// TIA Portal V17 export
// export: Created 2024-08-07T21:43:58.427102Z, ExportSetting WithDefaults, DisplayName Totally Integrated Automation Portal, DisplayVersion V17 Update 7, DisplayName TIA Portal Openness, DisplayVersion V17 Update 7, DisplayName TIA Portal Version Control Interface, DisplayVersion V17, DisplayName SINAMICS Startdrive Advanced, DisplayVersion V17 SP2, DisplayName SINAMICS Startdrive G110M, G120, G120C, G120D, G120P, G115D, DisplayVersion V17 SP2, DisplayName SINAMICS Startdrive G130, G150, S120, S150, SINAMICS MV, S210, DisplayVersion V17 SP2, DisplayName STEP 7 Professional, DisplayVersion V17 Update 7, DisplayName STEP 7 Safety, DisplayVersion V17 Update 6, DisplayName WinCC Advanced / Unified PC, DisplayVersion V17 Update 7
FUNCTION_BLOCK "READER_LOGIC"   // FB24, LAD
{ S7_Optimized_Access := 'TRUE' }
VERSION : 0.1
// stored: AutoNumber true, IsIECCheckEnabled false, IsRetainMemResEnabled false, MemoryReserve 100, SetENOAutomatically false, UDAEnableTagReadback false
   VAR_INPUT
      MODE : UInt;
      INIT_SCAN : Bool;
      SCAN_BUSY : Bool;
      SCAN_COMPLETE : Bool;
      STA_REC_1 : Bool;
      STA_REC : Bool;
      SCAN_OK1 : Bool;
      SCAN_OK2 : Bool;
      IJC_DISABLE : Bool;
      SCAN_LABEL : String;
      SCAN_POSITION : Int;
      SCAN_LEN : Int;
      READ_OF_SCAN : HW_SUBMODULE;
      NUM_OF_TUBE : Bool;
      RESET_SCANER : Bool;
   END_VAR
   VAR_OUTPUT
      REQUEST_SCAN : Bool;
      READ_STRG : String;
      SCAN_OK : Bool;
      MSG_STATUS_REQ : Bool;
      NFP_AUX : String;
      NFP_AUX2 : String;
      LECTURA_SCANER_ST : String;
      SCAN_CLEAR : Bool;
   END_VAR
   VAR
      RET_TRIG : IEC_TIMER;
   END_VAR
   VAR_TEMP
      ERROR_RECIBIDO_ESCANER : Int;
      RECIBIDO_SCANER : Array[0..254] of Char;
      RECIBIDO_SCANER_STRG : String;
      LECTURA_SCANER : String;
      done : Bool;
   END_VAR
   VAR_TEMP   // added for the SCL form of the ladder/FBD networks
      _w1 : Bool;
      _w2 : Bool;
      _w3 : Bool;
      _w4 : Bool;
      _w5 : Bool;
      _w6 : Bool;
   END_VAR
BEGIN

REGION Network 1
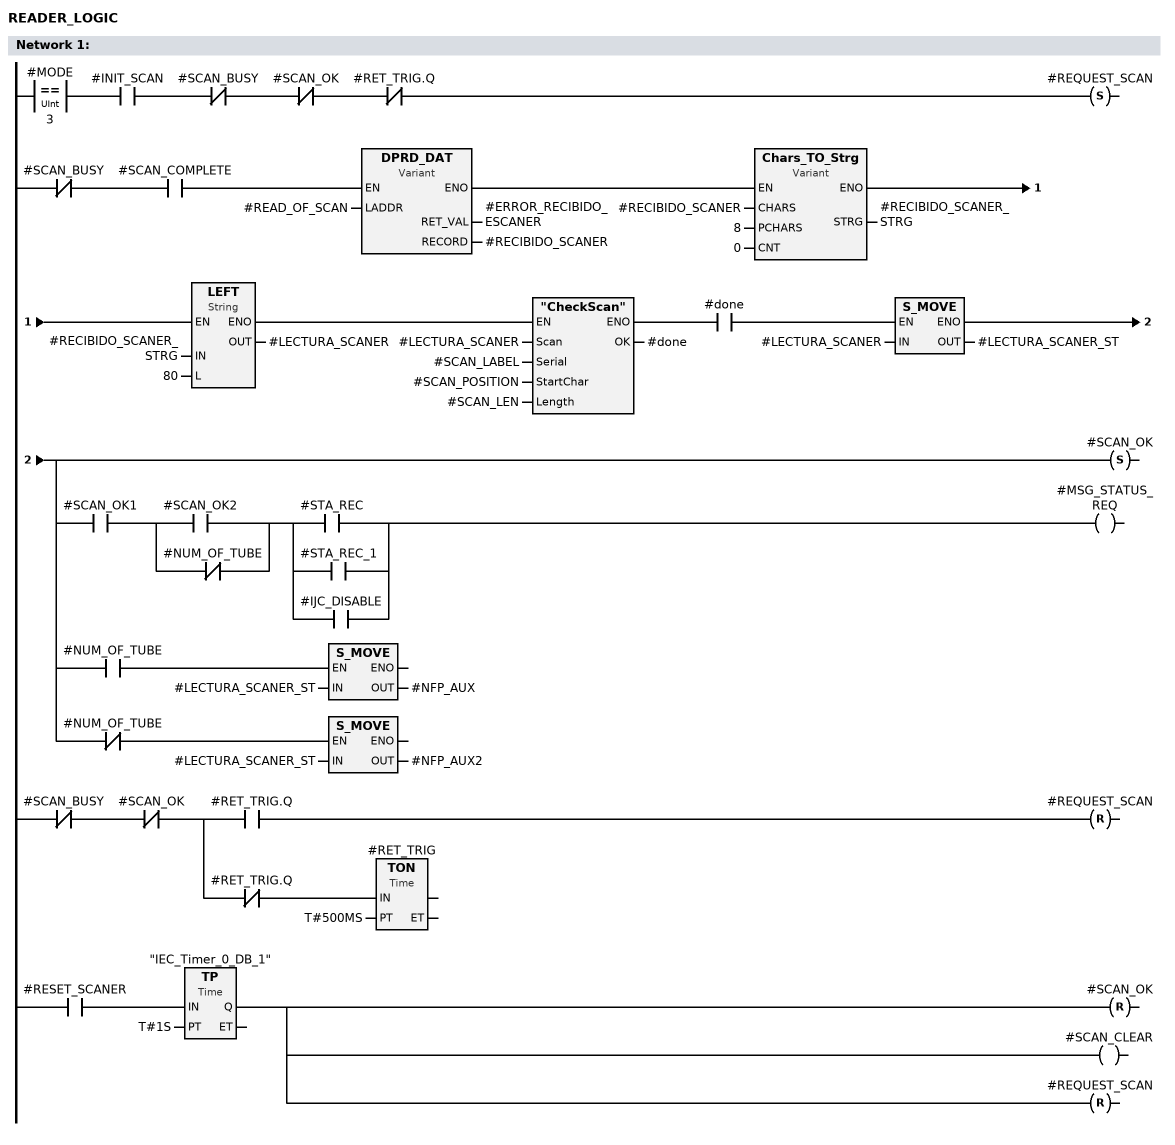
   RUNG wire#powerrail
      { S7_Templates := "SrcType := UInt" } EQ_Contact(in1 := #MODE, in2 := 3)
      Contact( #INIT_SCAN )
      I_Contact( #SCAN_BUSY )
      I_Contact( #SCAN_OK )
      I_Contact( #RET_TRIG.Q )
      S_Coil( #REQUEST_SCAN )
   END_RUNG
   RUNG wire#powerrail
      I_Contact( #SCAN_BUSY )
      Contact( #SCAN_COMPLETE )
      { S7_Templates := "[ptr_type := Variant, laddr_type := HW_IO]" } DPRD_DAT(LADDR := #READ_OF_SCAN, RET_VAL => #ERROR_RECIBIDO_ESCANER, RECORD => #RECIBIDO_SCANER)
      { S7_Templates := "[ptr_type := Variant, str_type := String]" } Chars_TO_Strg(Chars := #RECIBIDO_SCANER, pChars := 8, Cnt := 0, Strg => #RECIBIDO_SCANER_STRG)
      { S7_Templates := "str_type := String" } LEFT(IN := #RECIBIDO_SCANER_STRG, L := 80, OUT => #LECTURA_SCANER)
      "CheckScan"(Scan := #LECTURA_SCANER, Serial := #SCAN_LABEL, StartChar := #SCAN_POSITION, Length := #SCAN_LEN, OK => #done)
      Contact( #done )
      S_Move(in := #LECTURA_SCANER, out => #LECTURA_SCANER_ST)
      wire#w1
      S_Coil( #SCAN_OK )
   END_RUNG
   RUNG wire#w1
      Contact( #SCAN_OK1 )
      wire#w2
      Contact( #SCAN_OK2 )
      wire#w3
      Contact( #STA_REC )
      wire#w4
      Coil( #MSG_STATUS_REQ )
   END_RUNG
   RUNG wire#w2
      I_Contact( #NUM_OF_TUBE )
   END_RUNG wire#w3
   RUNG wire#w3
      Contact( #STA_REC_1 )
   END_RUNG wire#w4
   RUNG wire#w3
      Contact( #IJC_DISABLE )
   END_RUNG wire#w4
   RUNG wire#w1
      Contact( #NUM_OF_TUBE )
      S_Move(in := #LECTURA_SCANER_ST, out => #NFP_AUX)
   END_RUNG
   RUNG wire#w1
      I_Contact( #NUM_OF_TUBE )
      S_Move(in := #LECTURA_SCANER_ST, out => #NFP_AUX2)
   END_RUNG
   RUNG wire#powerrail
      I_Contact( #SCAN_BUSY )
      I_Contact( #SCAN_OK )
      wire#w5
      Contact( #RET_TRIG.Q )
      R_Coil( #REQUEST_SCAN )
   END_RUNG
   RUNG wire#w5
      I_Contact( #RET_TRIG.Q )
      { S7_Templates := "time_type := Time" } #RET_TRIG.TON(pt := T#500MS, et =>)
   END_RUNG
   RUNG wire#powerrail
      Contact( #RESET_SCANER )
      { S7_Templates := "time_type := Time" } "IEC_Timer_0_DB_1".TP(pt := T#1S, et =>)
      wire#w6
      R_Coil( #SCAN_OK )
   END_RUNG
   RUNG wire#w6
      Coil( #SCAN_CLEAR )
   END_RUNG
   RUNG wire#w6
      R_Coil( #REQUEST_SCAN )
   END_RUNG
   // the same network as SCL:
   IF (#MODE = 3) AND #INIT_SCAN AND NOT #SCAN_BUSY AND NOT #SCAN_OK AND NOT #RET_TRIG.Q THEN
       #REQUEST_SCAN := TRUE;
   END_IF;
   #ERROR_RECIBIDO_ESCANER := DPRD_DAT(EN := NOT #SCAN_BUSY AND #SCAN_COMPLETE,
                           LADDR := #READ_OF_SCAN,
                           RECORD => #RECIBIDO_SCANER,
                           ENO => #_w1);
   Chars_TO_Strg(EN := #_w1,
                 Chars := #RECIBIDO_SCANER,
                 pChars := 8,
                 Cnt := 0,
                 Strg => #RECIBIDO_SCANER_STRG,
                 ENO => #_w2);
   LEFT(EN := #_w2, IN := #RECIBIDO_SCANER_STRG, L := 80, OUT => #LECTURA_SCANER, ENO => #_w3);
   "CheckScan"(EN := #_w3,
               Scan := #LECTURA_SCANER,
               Serial := #SCAN_LABEL,
               StartChar := #SCAN_POSITION,
               Length := #SCAN_LEN,
               OK => #done,
               ENO => #_w4);
   #_w5 := #_w4 AND #done;
   IF #_w5 THEN
       #LECTURA_SCANER_ST := #LECTURA_SCANER;
       #SCAN_OK := TRUE;
   END_IF;
   #MSG_STATUS_REQ := #_w5 AND #SCAN_OK1 AND (#SCAN_OK2 OR NOT #NUM_OF_TUBE) AND (#STA_REC OR #STA_REC_1 OR #IJC_DISABLE);
   IF #_w5 AND #NUM_OF_TUBE THEN #NFP_AUX := #LECTURA_SCANER_ST; END_IF;
   IF #_w5 AND NOT #NUM_OF_TUBE THEN #NFP_AUX2 := #LECTURA_SCANER_ST; END_IF;
   #_w6 := NOT #SCAN_BUSY AND NOT #SCAN_OK;
   IF #_w6 AND #RET_TRIG.Q THEN #REQUEST_SCAN := FALSE; END_IF;
   #RET_TRIG.TON(IN := #_w6 AND NOT #RET_TRIG.Q, PT := T#500MS);
   "IEC_Timer_0_DB_1".TP(IN := #RESET_SCANER, PT := T#1S);
   IF "IEC_Timer_0_DB_1".Q THEN #SCAN_OK := FALSE; END_IF;
   #SCAN_CLEAR := "IEC_Timer_0_DB_1".Q;
   IF "IEC_Timer_0_DB_1".Q THEN #REQUEST_SCAN := FALSE; END_IF;
END_REGION
END_FUNCTION_BLOCK
